PROGRAM MAIN
VAR
END_VAR

;

END_PROGRAM

(* stored: Version 1.1.0.1, ProductVersion 3.1.0.36
   POU MAIN: Id {e6c5d348-b58a-45c9-80d1-f4c01767d25a}, SpecialFunc None *)
